FUNCTION_BLOCK LoadCell
VAR_INPUT
	LoadCellInput : LoadCellI;
END_VAR
VAR_OUTPUT
	LoadCellOutput : LoadCellO;
END_VAR
VAR
	ScaleComp : itfScaleAnalogInputImplement;
	Scale : itfScale;
END_VAR

Map();
Scale.mScale();

METHOD PRIVATE Map : BOOL
VAR_INPUT
END_VAR
Scale := ScaleComp;
Scale.pAnalogSignal := LoadCellInput.AnalogSignal;
Scale.pMaxSignalValue := LoadCellInput.MaxSignalValue;
Scale.pMaxUnitValue := LoadCellInput.MaxUnitValue;

LoadCellOutput.ScaledValue :=Scale.pScaledSignal;
END_METHOD

END_FUNCTION_BLOCK

(* stored: Version 1.1.0.1, ProductVersion 3.1.4024.12
   POU LoadCell: Id {57e1b19f-4784-4442-b316-20a78cd83725}, SpecialFunc None
   Method Map: Id {7a545051-e34e-40a3-82c2-e64eeaf805cb} *)
